% RSLogix 500 project MLO3B JOB 5.3.RSS, saved by version 10.00.00.00 %
PROJECT "MLO3B"    % processor: Bul.1763 MicroLogix 1100 Series B %

PROGRAM FILES
  LAD 2   4 rungs

DATA FILES
  O0 OUTPUT  4 elements
  I1 INPUT  6 elements
  S2 STATUS  66 elements
  B3 BINARY  1 elements
  T4 TIMER  1 elements
  C5 COUNTER  1 elements
  R6 CONTROL  1 elements
  N7 INTEGER  1 elements
  F8 FLOAT  1 elements

LADDER 2
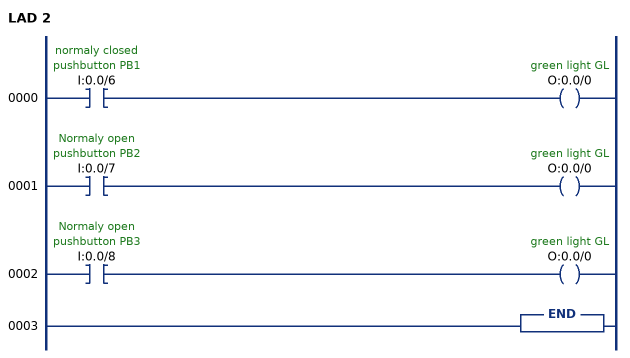
% Rung: 0 %
SOR XIC I:0.0/6 OTE O:0.0/0 EOR
%   I:0.0/6  PB1  "normaly closed pushbutton" %
%   O:0.0/0  GL  "green light" %
% Rung: 1 %
SOR XIC I:0.0/7 OTE O:0.0/0 EOR
%   I:0.0/7  PB2  "Normaly open pushbutton" %
%   O:0.0/0  GL  "green light" %
% Rung: 2 %
SOR XIC I:0.0/8 OTE O:0.0/0 EOR
%   I:0.0/8  PB3  "Normaly open pushbutton" %
%   O:0.0/0  GL  "green light" %
% Rung: 3 %
SOR END EOR

OTHER DOCUMENTED ADDRESSES
  I:0.0/0  ES  "Emergcy stop"
  I:0.0/1  CR1C  "Control relay 1 contacts"
  I:0.0/2  CR2C  "Control realy 2 contacts"
  I:0.0/3  3PSSA  "Three position selector switch a position"
  I:0.0/4  3PSSB  "Three postion selector switch b"
  I:0.0/5  2PSS  "Two postion selector switch"
  IOS  
  O:0.0/1  YL  "Yellow light"
  O:0.0/2  RL  "Red light"
  O:0.0/3  BL  "Blue light"
  O:0.0/4  CR1  "Control relay 1"
  O:0.0/5  CR2  "Control relay 2"
  O:0.0/6  GREEN_LIGHT
